{attribute 'qualified_only'}
VAR_GLOBAL
END_VAR

(* stored: Version 1.1.0.1, ProductVersion 3.1.4024.16
   GVL Global_1: Id {f2782c1c-46e7-4746-a584-b9e27c30a18f} *)
